DATA_BLOCK "DB_ProcessSlots"
{ S7_Optimized_Access := 'TRUE' }
VERSION : 0.1
// ATTRIBUTES
// AUTO_NUMBER = False
// BLOCK_NUMBER = 2600
// END_ATTRIBUTES
   VAR
      Slots : Array[1..16] of "UDT_ProcessSlot";
   END_VAR


BEGIN
   Slots[1].SlotID := 1;
   Slots[1].PositionTag := 'A_ScanRotate';
   Slots[2].SlotID := 2;
   Slots[2].PositionTag := 'F_Robot1Grip1';
   Slots[3].SlotID := 3;
   Slots[3].PositionTag := 'F_Robot1Grip2';
   Slots[4].SlotID := 4;
   Slots[4].PositionTag := 'B_Press1';
   Slots[5].SlotID := 5;
   Slots[5].PositionTag := 'C_Glue';
   Slots[6].SlotID := 6;
   Slots[6].PositionTag := 'F_Robot2Grip1';
   Slots[7].SlotID := 7;
   Slots[7].PositionTag := 'F_Robot2Grip2';
   Slots[8].SlotID := 8;
   Slots[8].PositionTag := 'C_GlueNGBuffer';
   Slots[9].SlotID := 9;
   Slots[9].PositionTag := 'C_MagnScanNGBuffer';
   Slots[10].SlotID := 10;
   Slots[10].PositionTag := 'B_Press2';
   Slots[11].SlotID := 11;
   Slots[11].PositionTag := 'F_Robot3Grip1';
   Slots[12].SlotID := 12;
   Slots[12].PositionTag := 'F_Robot3Grip2';
   Slots[13].SlotID := 13;
   Slots[13].PositionTag := 'H_ShafeLine';
   Slots[14].SlotID := 14;
   Slots[14].PositionTag := 'J_ShafeLine';
   Slots[15].SlotID := 15;
   Slots[15].PositionTag := 'K_ShafeLine';
   Slots[16].SlotID := 16;
   Slots[16].PositionTag := 'L_ShafeLine';

END_DATA_BLOCK

